PROGRAM PMPS
VAR
	fbArbiterIO : FB_SubSysToArbiter_IO;
	bRemove: BOOL;
	bExist: BOOL;
	ID: UDINT;
END_VAR

(*FastFaultOuput*)
g_FastFaultOutput1.Execute(bAutoReset:= TRUE);
g_FastFaultOutput2.Execute(i_xVeto:=PMPS_GVL.stCurrentBeamParameters.aStoppers[K_Stopper.ST3K4], bAutoReset:= TRUE);

fbArbiterIO(Arbiter := g_fbArbiter1, fbFFHWO := g_FastFaultOutput1);

bExist:= g_fbArbiter1.CheckRequestInPool(ID);
if (bRemove) THEN
	g_fbArbiter1.RemoveRequest(ID);
END_IF

END_PROGRAM

(* stored: Version 1.1.0.1, ProductVersion 3.1.4022.18
   POU PMPS: Id {354279ff-d518-454c-b9bb-5f6640e67b86}, SpecialFunc None *)
